FUNCTION_BLOCK xscal_fi
VAR_INPUT
    a: LREAL;
    ix0: DINT;
END_VAR
VAR_IN_OUT
    x: ARRAY [0..29] OF LREAL;
END_VAR
VAR_TEMP
    k: DINT;
END_VAR

k := ix0;
WHILE k <= (ix0 + 5) DO
    x[k - 1] := x[k - 1] * a;
    k := k + 1;
END_WHILE;

END_FUNCTION_BLOCK

(* stored: Version 1.1.0.1, ProductVersion 3.1.4024.12
   POU xscal_fi: Id {23c6bca1-0067-43e1-b664-28cb591140b4}, SpecialFunc None *)
